(*
version 1.1	10. mar. 2009
programmer 	hugo
tested by		tobias

this function calculates the inverse erf (error) function.

*)
FUNCTION ERFC : REAL
VAR_INPUT
	X : REAL;
END_VAR

ERFC := 1.0 - ERF(X);

(* revision history
hm	7. apr. 2008	rev 1.0
	original version

hm	10. mar. 2009	rev 1.1
	real constants updated to new systax using dot

*)

END_FUNCTION

(* stored: Version 1.1.0.1
   POU ERFC: Id {d16983be-2e46-4790-9707-f8f05f7233f3}, SpecialFunc None *)
